Fanuc TP program (LS listing): second_power_source.ls

/PROG move
/ATTR
/MN
:UFRAME=5;
:UTOOL_NUM=6;
:
:LBL[1];
:PR[100,1]=$SCR_GRP[1].$MCH_POS_X+R[101];
:PR[100,2]=$SCR_GRP[1].$MCH_POS_Y+R[102];
:PR[100,3]=$SCR_GRP[1].$MCH_POS_Z+R[103];
:
:L PR[100] WELD_SPEED CNT100 COORD PTH;
:R[111]=PR[100,1];
:R[112]=PR[100,2];
:R[113]=PR[100,3];
:JMP LBL[1];
:
/POS
/END
